FUNCTION_BLOCK FB_DriveInterface
VAR_INPUT
END_VAR
VAR_OUTPUT
END_VAR
VAR
	power: MC_Power; //MC_Power instance
	reset: MC_Reset;
	moveabs: MC_MoveAbsolute;
END_VAR

VAR_IN_OUT
	plcAxis:typeDriveInterface; //axis ref to the rest of PLC
	ncAxis:axis_ref; //axis ref of the NC drive (only beckhoff)
	
END_VAR

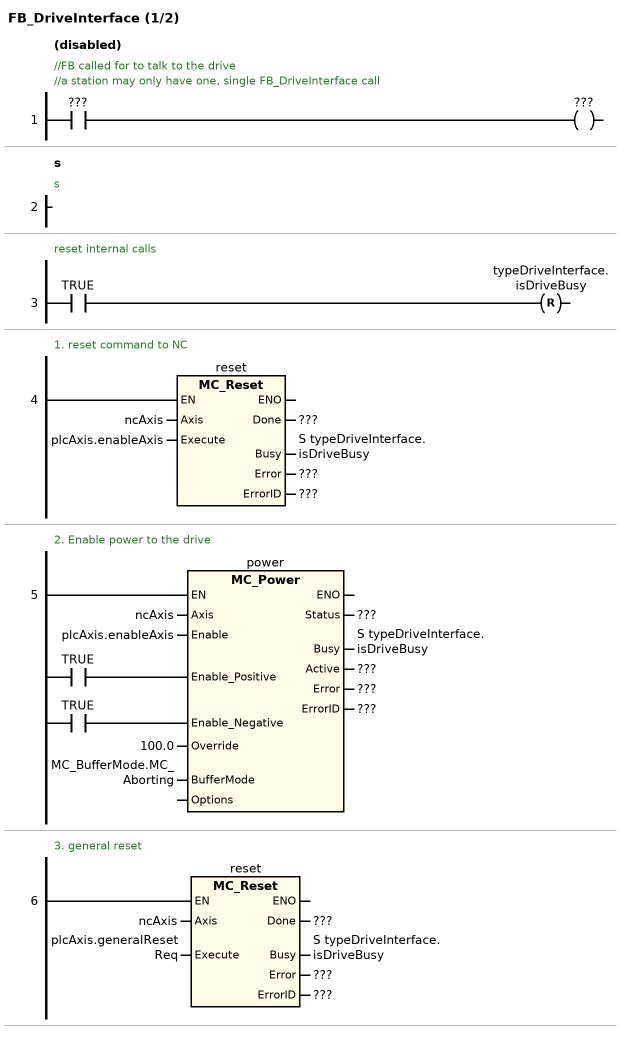
// NETWORK 1 (disabled)
// //FB called for to talk to the drive
// //a station may only have one, single FB_DriveInterface call
// ??? := ???;

// NETWORK 2: s
// s

// NETWORK 3
// reset internal calls
typeDriveInterface.isDriveBusy R= TRUE;

// NETWORK 4
// 1. reset command to NC
reset(Axis := ncAxis, Execute := plcAxis.enableAxis); // MC_Reset
typeDriveInterface.isDriveBusy S= reset.Busy;

// NETWORK 5
// 2. Enable power to the drive
power(
    Axis := ncAxis,
    Enable := plcAxis.enableAxis,
    Enable_Positive := TRUE,
    Enable_Negative := TRUE,
    Override := 100.0,
    BufferMode := MC_BufferMode.MC_Aborting); // MC_Power
typeDriveInterface.isDriveBusy S= power.Busy;

// NETWORK 6
// 3. general reset
reset(Axis := ncAxis, Execute := plcAxis.generalResetReq); // MC_Reset
typeDriveInterface.isDriveBusy S= reset.Busy;

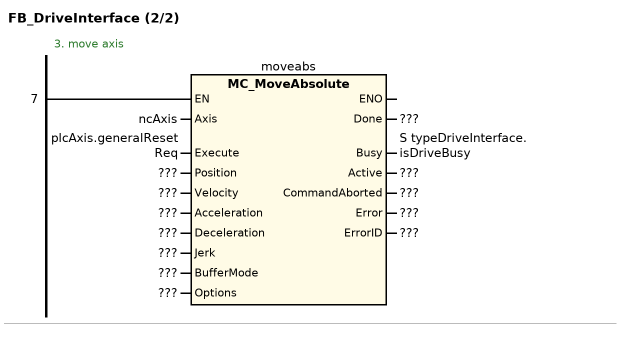
// NETWORK 7
// 3. move axis
moveabs(Axis := ncAxis, Execute := plcAxis.generalResetReq); // MC_MoveAbsolute
typeDriveInterface.isDriveBusy S= moveabs.Busy;

END_FUNCTION_BLOCK

(* stored: Version 1.1.0.1, ProductVersion 3.1.4024.12
   POU FB_DriveInterface: Id {ef5a2760-99ed-4752-b6d0-8e47bd4f419b}, SpecialFunc None *)
